// TIA Portal V18 export
// export: Created 2000-01-01T00:00:00.0000000Z, ExportSetting None
VAR_GLOBAL   // PLC tag table "Motor_Basic_IO"
   DI_StartPB AT %I0.0 : Bool;
   DI_StopPB AT %I0.1 : Bool;
   DI_Fault AT %I0.2 : Bool;
   DO_MotorRun AT %Q0.0 : Bool;
END_VAR
